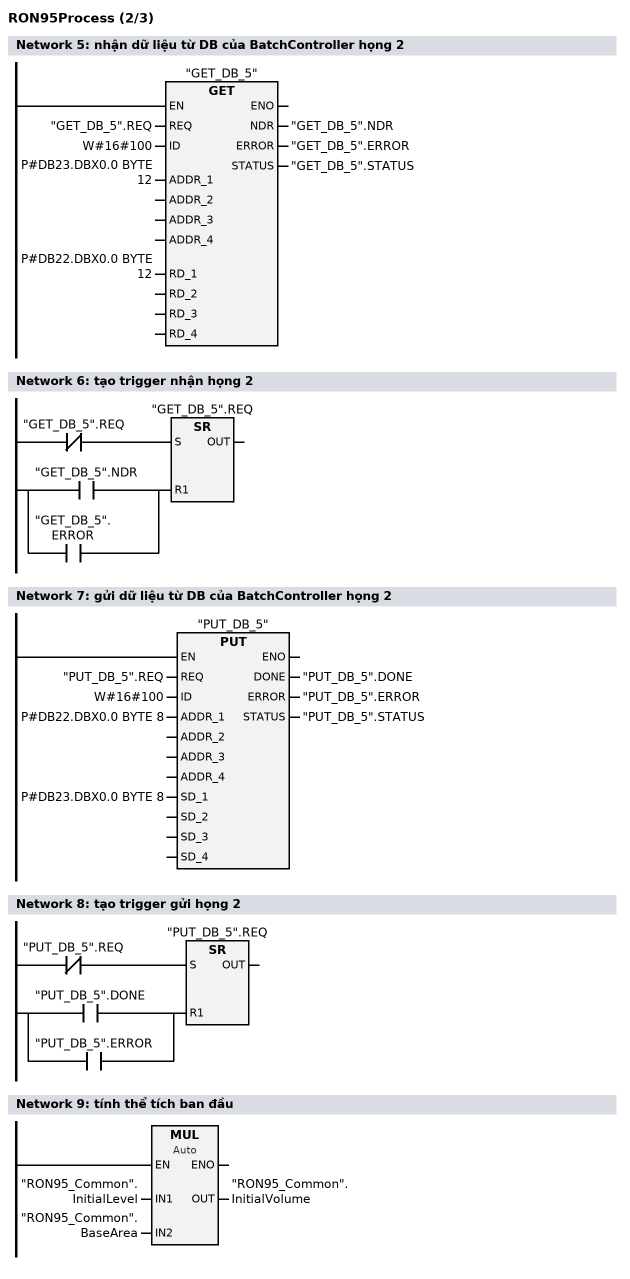
   "GET_DB_5"(REQ := "GET_DB_5".REQ,   // GET
              ID := W#16#100,
              ADDR_1 := P#DB23.DBX0.0 BYTE 12,
              RD_1 := P#DB22.DBX0.0 BYTE 12,
              NDR => "GET_DB_5".NDR,
              ERROR => "GET_DB_5".ERROR,
              STATUS => "GET_DB_5".STATUS);
END_REGION

REGION Network 6: tạo trigger nhận họng 2
   RUNG wire#powerrail
      I_Contact( "GET_DB_5".REQ )
      S_SR(operand := "GET_DB_5".REQ, r1 := wire#w1)
   END_RUNG
   RUNG wire#powerrail
      Contact( "GET_DB_5".NDR )
   END_RUNG wire#w1
   RUNG wire#powerrail
      Contact( "GET_DB_5".ERROR )
   END_RUNG wire#w1
   // the same network as SCL:
   IF NOT "GET_DB_5".REQ THEN
       "GET_DB_5".REQ := TRUE;   // SR flip-flop
   END_IF;
   IF "GET_DB_5".NDR OR "GET_DB_5".ERROR THEN "GET_DB_5".REQ := FALSE; END_IF;
END_REGION

REGION Network 7: gửi dữ liệu từ DB của BatchController họng 2
   "PUT_DB_5"(REQ := "PUT_DB_5".REQ,   // PUT
              ID := W#16#100,
              ADDR_1 := P#DB22.DBX0.0 BYTE 8,
              SD_1 := P#DB23.DBX0.0 BYTE 8,
              DONE => "PUT_DB_5".DONE,
              ERROR => "PUT_DB_5".ERROR,
              STATUS => "PUT_DB_5".STATUS);
END_REGION

REGION Network 8: tạo trigger gửi họng 2
   RUNG wire#powerrail
      I_Contact( "PUT_DB_5".REQ )
      S_SR(operand := "PUT_DB_5".REQ, r1 := wire#w1)
   END_RUNG
   RUNG wire#powerrail
      Contact( "PUT_DB_5".DONE )
   END_RUNG wire#w1
   RUNG wire#powerrail
      Contact( "PUT_DB_5".ERROR )
   END_RUNG wire#w1
   // the same network as SCL:
   IF NOT "PUT_DB_5".REQ THEN
       "PUT_DB_5".REQ := TRUE;   // SR flip-flop
   END_IF;
   IF "PUT_DB_5".DONE OR "PUT_DB_5".ERROR THEN "PUT_DB_5".REQ := FALSE; END_IF;
END_REGION

REGION Network 9: tính thể tích ban đầu
   RUNG wire#powerrail
      Mul(in1 := "RON95_Common".InitialLevel, in2 := "RON95_Common".BaseArea, out => "RON95_Common".InitialVolume)
   END_RUNG
   // the same network as SCL:
   "RON95_Common".InitialVolume := "RON95_Common".InitialLevel * "RON95_Common".BaseArea;
END_REGION

REGION Network 10: tính thể tích hiện tại
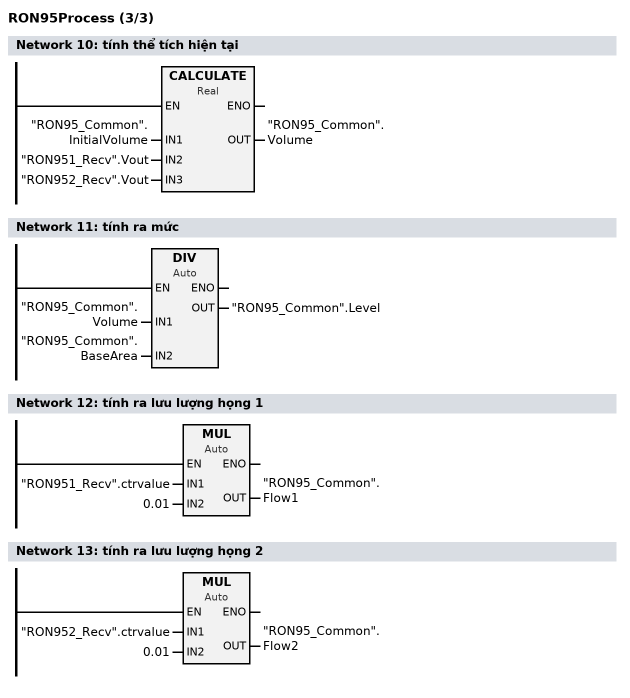
   RUNG wire#powerrail
      { S7_Templates := "SrcType := Real"; S7_Expression := "IN1-IN2-IN3" } Calculate(in1 := "RON95_Common".InitialVolume, in2 := "RON951_Recv".Vout, in3 := "RON952_Recv".Vout, out => "RON95_Common".Volume)
   END_RUNG
   // the same network as SCL:
   "RON95_Common".Volume := "RON95_Common".InitialVolume-"RON951_Recv".Vout-"RON952_Recv".Vout;
END_REGION

REGION Network 11: tính ra mức
   RUNG wire#powerrail
      Div(in1 := "RON95_Common".Volume, in2 := "RON95_Common".BaseArea, out => "RON95_Common".Level)
   END_RUNG
   // the same network as SCL:
   "RON95_Common".Level := "RON95_Common".Volume / "RON95_Common".BaseArea;
END_REGION

REGION Network 12: tính ra lưu lượng họng 1
   RUNG wire#powerrail
      Mul(in1 := "RON951_Recv".ctrvalue, in2 := 0.01, out => "RON95_Common".Flow1)
   END_RUNG
   // the same network as SCL:
   "RON95_Common".Flow1 := "RON951_Recv".ctrvalue * 0.01;
END_REGION

REGION Network 13: tính ra lưu lượng họng 2
   RUNG wire#powerrail
      Mul(in1 := "RON952_Recv".ctrvalue, in2 := 0.01, out => "RON95_Common".Flow2)
   END_RUNG
   // the same network as SCL:
   "RON95_Common".Flow2 := "RON952_Recv".ctrvalue * 0.01;
END_REGION
END_FUNCTION

FUNCTION "E5Process" : Void   // FC4, LAD
{ S7_Optimized_Access := 'TRUE' }
VERSION : 0.1
BEGIN

REGION Network 1: nhận dữ liệu từ DB của BatchController họng 1
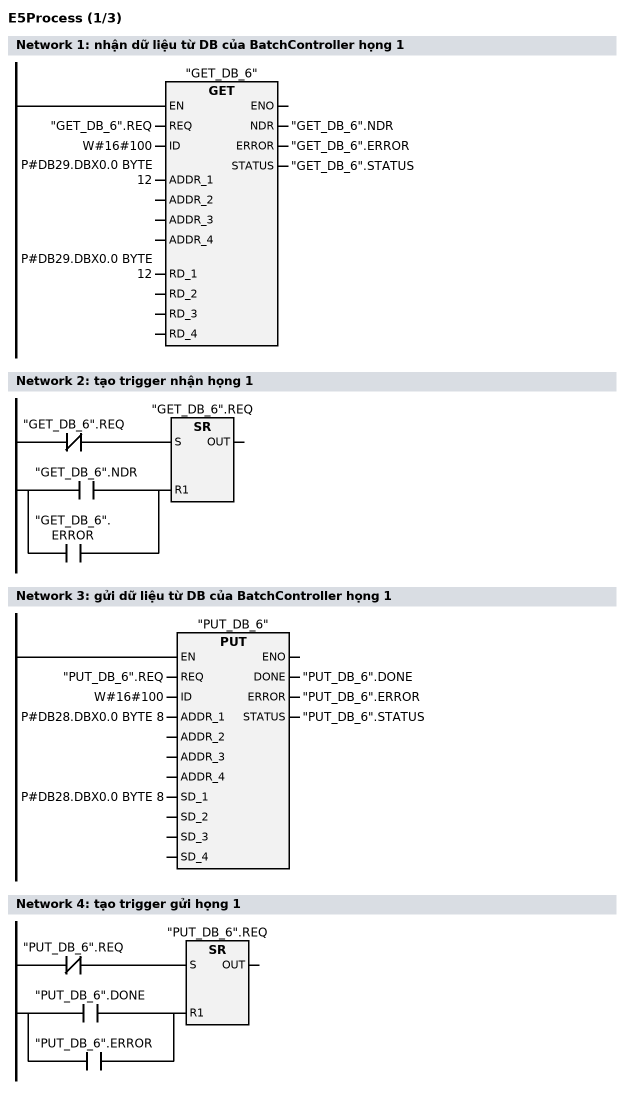
   "GET_DB_6"(REQ := "GET_DB_6".REQ,   // GET
              ID := W#16#100,
              ADDR_1 := P#DB29.DBX0.0 BYTE 12,
              RD_1 := P#DB29.DBX0.0 BYTE 12,
              NDR => "GET_DB_6".NDR,
              ERROR => "GET_DB_6".ERROR,
              STATUS => "GET_DB_6".STATUS);
END_REGION

REGION Network 2: tạo trigger nhận họng 1
   RUNG wire#powerrail
      I_Contact( "GET_DB_6".REQ )
      S_SR(operand := "GET_DB_6".REQ, r1 := wire#w1)
   END_RUNG
   RUNG wire#powerrail
      Contact( "GET_DB_6".NDR )
   END_RUNG wire#w1
   RUNG wire#powerrail
      Contact( "GET_DB_6".ERROR )
   END_RUNG wire#w1
   // the same network as SCL:
   IF NOT "GET_DB_6".REQ THEN
       "GET_DB_6".REQ := TRUE;   // SR flip-flop
   END_IF;
   IF "GET_DB_6".NDR OR "GET_DB_6".ERROR THEN "GET_DB_6".REQ := FALSE; END_IF;
END_REGION

REGION Network 3: gửi dữ liệu từ DB của BatchController họng 1
   "PUT_DB_6"(REQ := "PUT_DB_6".REQ,   // PUT
              ID := W#16#100,
              ADDR_1 := P#DB28.DBX0.0 BYTE 8,
              SD_1 := P#DB28.DBX0.0 BYTE 8,
              DONE => "PUT_DB_6".DONE,
              ERROR => "PUT_DB_6".ERROR,
              STATUS => "PUT_DB_6".STATUS);
END_REGION

REGION Network 4: tạo trigger gửi họng 1
   RUNG wire#powerrail
      I_Contact( "PUT_DB_6".REQ )
      S_SR(operand := "PUT_DB_6".REQ, r1 := wire#w1)
   END_RUNG
   RUNG wire#powerrail
      Contact( "PUT_DB_6".DONE )
   END_RUNG wire#w1
   RUNG wire#powerrail
      Contact( "PUT_DB_6".ERROR )
   END_RUNG wire#w1
   // the same network as SCL:
   IF NOT "PUT_DB_6".REQ THEN
       "PUT_DB_6".REQ := TRUE;   // SR flip-flop
   END_IF;
   IF "PUT_DB_6".DONE OR "PUT_DB_6".ERROR THEN "PUT_DB_6".REQ := FALSE; END_IF;
END_REGION

REGION Network 5: nhận dữ liệu từ DB của BatchController họng 2
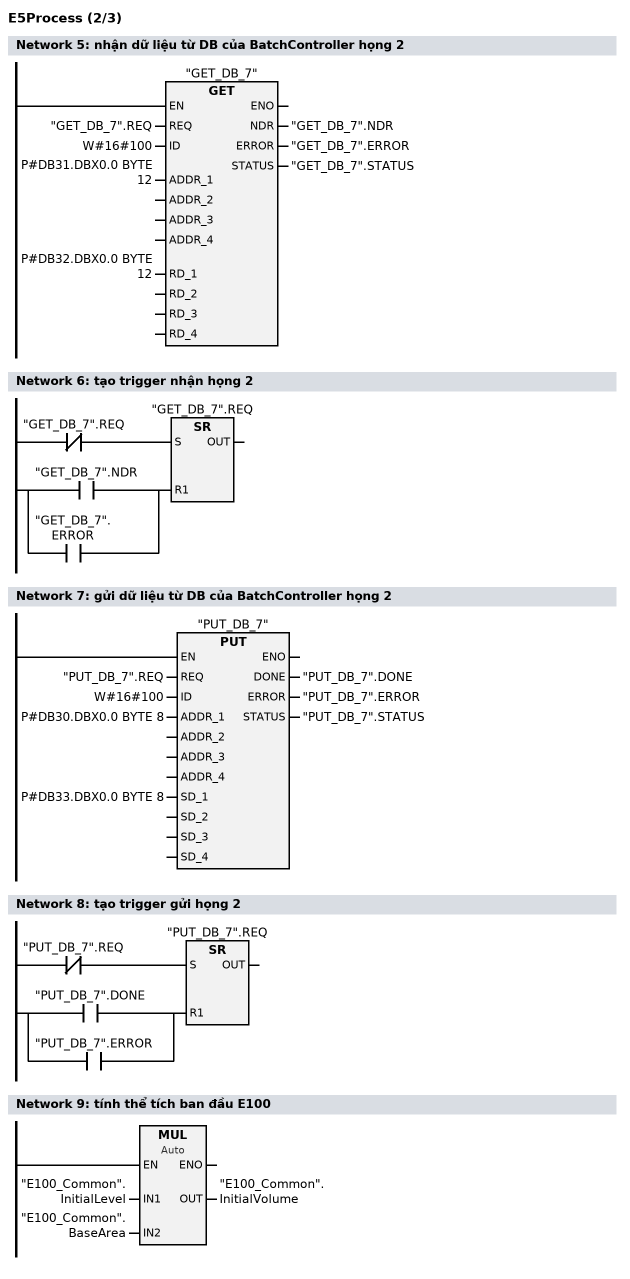
   "GET_DB_7"(REQ := "GET_DB_7".REQ,   // GET
              ID := W#16#100,
              ADDR_1 := P#DB31.DBX0.0 BYTE 12,
              RD_1 := P#DB32.DBX0.0 BYTE 12,
              NDR => "GET_DB_7".NDR,
              ERROR => "GET_DB_7".ERROR,
              STATUS => "GET_DB_7".STATUS);
END_REGION

REGION Network 6: tạo trigger nhận họng 2
   RUNG wire#powerrail
      I_Contact( "GET_DB_7".REQ )
      S_SR(operand := "GET_DB_7".REQ, r1 := wire#w1)
   END_RUNG
   RUNG wire#powerrail
      Contact( "GET_DB_7".NDR )
   END_RUNG wire#w1
   RUNG wire#powerrail
      Contact( "GET_DB_7".ERROR )
   END_RUNG wire#w1
   // the same network as SCL:
   IF NOT "GET_DB_7".REQ THEN
       "GET_DB_7".REQ := TRUE;   // SR flip-flop
   END_IF;
   IF "GET_DB_7".NDR OR "GET_DB_7".ERROR THEN "GET_DB_7".REQ := FALSE; END_IF;
END_REGION

REGION Network 7: gửi dữ liệu từ DB của BatchController họng 2
   "PUT_DB_7"(REQ := "PUT_DB_7".REQ,   // PUT
              ID := W#16#100,
              ADDR_1 := P#DB30.DBX0.0 BYTE 8,
              SD_1 := P#DB33.DBX0.0 BYTE 8,
              DONE => "PUT_DB_7".DONE,
              ERROR => "PUT_DB_7".ERROR,
              STATUS => "PUT_DB_7".STATUS);
END_REGION

REGION Network 8: tạo trigger gửi họng 2
   RUNG wire#powerrail
      I_Contact( "PUT_DB_7".REQ )
      S_SR(operand := "PUT_DB_7".REQ, r1 := wire#w1)
   END_RUNG
   RUNG wire#powerrail
      Contact( "PUT_DB_7".DONE )
   END_RUNG wire#w1
   RUNG wire#powerrail
      Contact( "PUT_DB_7".ERROR )
   END_RUNG wire#w1
   // the same network as SCL:
   IF NOT "PUT_DB_7".REQ THEN
       "PUT_DB_7".REQ := TRUE;   // SR flip-flop
   END_IF;
   IF "PUT_DB_7".DONE OR "PUT_DB_7".ERROR THEN "PUT_DB_7".REQ := FALSE; END_IF;
END_REGION

REGION Network 9: tính thể tích ban đầu E100
   RUNG wire#powerrail
      Mul(in1 := "E100_Common".InitialLevel, in2 := "E100_Common".BaseArea, out => "E100_Common".InitialVolume)
   END_RUNG
   // the same network as SCL:
   "E100_Common".InitialVolume := "E100_Common".InitialLevel * "E100_Common".BaseArea;
END_REGION

REGION Network 10: tính thể tích hiện tại E100
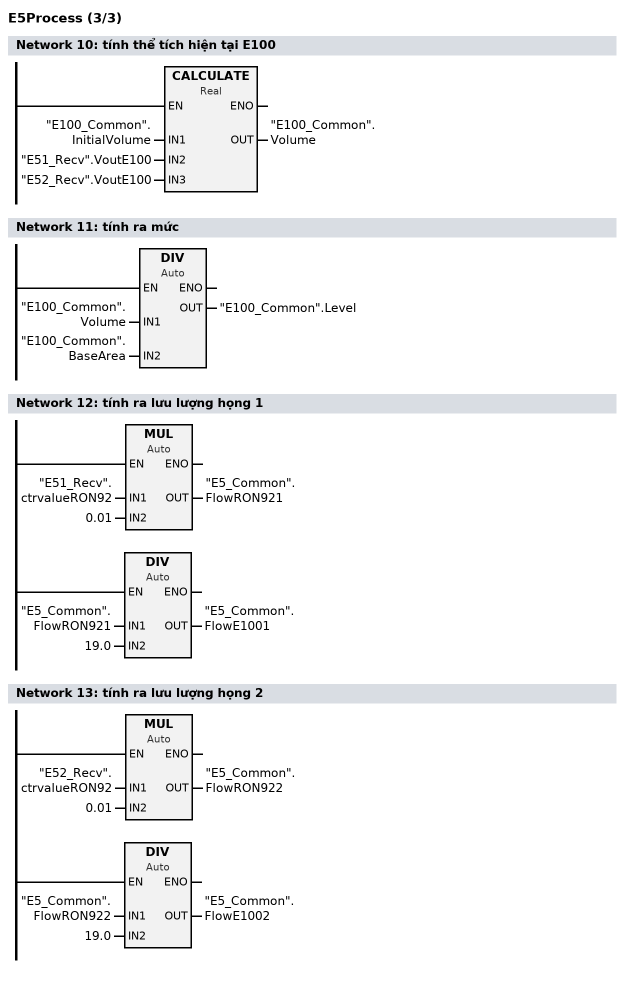
   RUNG wire#powerrail
      { S7_Templates := "SrcType := Real"; S7_Expression := "IN1-IN2-IN3" } Calculate(in1 := "E100_Common".InitialVolume, in2 := "E51_Recv".VoutE100, in3 := "E52_Recv".VoutE100, out => "E100_Common".Volume)
   END_RUNG
   // the same network as SCL:
   "E100_Common".Volume := "E100_Common".InitialVolume-"E51_Recv".VoutE100-"E52_Recv".VoutE100;
END_REGION

REGION Network 11: tính ra mức
   RUNG wire#powerrail
      Div(in1 := "E100_Common".Volume, in2 := "E100_Common".BaseArea, out => "E100_Common".Level)
   END_RUNG
   // the same network as SCL:
   "E100_Common".Level := "E100_Common".Volume / "E100_Common".BaseArea;
END_REGION

REGION Network 12: tính ra lưu lượng họng 1
   RUNG wire#powerrail
      Mul(in1 := "E51_Recv".ctrvalueRON92, in2 := 0.01, out => "E5_Common".FlowRON921)
   END_RUNG
   RUNG wire#powerrail
      Div(in1 := "E5_Common".FlowRON921, in2 := 19.0, out => "E5_Common".FlowE1001)
   END_RUNG
   // the same network as SCL:
   "E5_Common".FlowRON921 := "E51_Recv".ctrvalueRON92 * 0.01;
   "E5_Common".FlowE1001 := "E5_Common".FlowRON921 / 19.0;
END_REGION

REGION Network 13: tính ra lưu lượng họng 2
   RUNG wire#powerrail
      Mul(in1 := "E52_Recv".ctrvalueRON92, in2 := 0.01, out => "E5_Common".FlowRON922)
   END_RUNG
   RUNG wire#powerrail
      Div(in1 := "E5_Common".FlowRON922, in2 := 19.0, out => "E5_Common".FlowE1002)
   END_RUNG
   // the same network as SCL:
   "E5_Common".FlowRON922 := "E52_Recv".ctrvalueRON92 * 0.01;
   "E5_Common".FlowE1002 := "E5_Common".FlowRON922 / 19.0;
END_REGION
END_FUNCTION

ORGANIZATION_BLOCK "Main"   // OB1, LAD, ProgramCycle
TITLE = "Main Program Sweep (Cycle)"
{ S7_Optimized_Access := 'TRUE' }
VERSION : 0.1
   VAR_INPUT
      Initial_Call : Bool;   // Initial call of this OB
      Remanence : Bool;   // =True, if remanent data are available
   END_VAR
BEGIN

REGION Network 1: Chương trình xử lý của Diezel
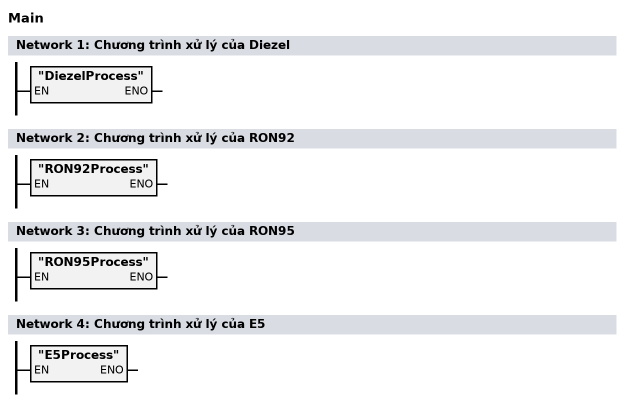
   RUNG wire#powerrail
      "DiezelProcess"()
   END_RUNG
   // the same network as SCL:
   "DiezelProcess"();
END_REGION

REGION Network 2: Chương trình xử lý của RON92
   RUNG wire#powerrail
      "RON92Process"()
   END_RUNG
   // the same network as SCL:
   "RON92Process"();
END_REGION

REGION Network 3: Chương trình xử lý của RON95
   RUNG wire#powerrail
      "RON95Process"()
   END_RUNG
   // the same network as SCL:
   "RON95Process"();
END_REGION

REGION Network 4: Chương trình xử lý của E5
   RUNG wire#powerrail
      "E5Process"()
   END_RUNG
   // the same network as SCL:
   "E5Process"();
END_REGION
END_ORGANIZATION_BLOCK